// TIA Portal project "TaskCiclico" (V16)

(* hardware
DEVICE "S7-1200 station_1"  S7-1200 Station
   slot 0: "Telaio di montaggio_0"  S7-1200 Rack  Rack  V1.0
   slot 1: "PLC_1"  CPU 1214C DC/DC/DC  6ES7 214-1AG40-0XB0  V4.1
*)

// ===== PLC "PLC_1"  CPU 1214C DC/DC/DC =====

VAR_GLOBAL   // PLC tag table "Tabella delle variabili standard"
   "Reset" AT %I0.0 : Bool;
END_VAR

DATA_BLOCK "VariabiliGlobali"   // DB1
{ S7_Optimized_Access := 'TRUE' }
VERSION : 0.1
   VAR RETAIN
      Signal : Real;
      DelayedSignal : Real;
      N_SMP : Int := 5;
      SignalThreshold : Real := 40.0;
   END_VAR
BEGIN
END_DATA_BLOCK

DATA_BLOCK "FB_Shift_DB"   // DB2
{ S7_Optimized_Access := 'TRUE' }
VERSION : 0.1
// stored: InstanceOfName FB_Shift
"FB_Shift"
BEGIN
END_DATA_BLOCK

FUNCTION_BLOCK "FB_Shift"   // FB1, LAD
{ S7_Optimized_Access := 'TRUE' }
VERSION : 0.1
   VAR_INPUT
      Ingresso : Real;
      N_SMP : Int;
      Restart : Bool;
   END_VAR
   VAR_OUTPUT
      Uscita : Real;
   END_VAR
   VAR RETAIN
      STORE : Array[0..19] of Real;
      indice_1 : Int;
      indice_2 : Int;
      sup : Int;
   END_VAR
BEGIN

REGION Network 1
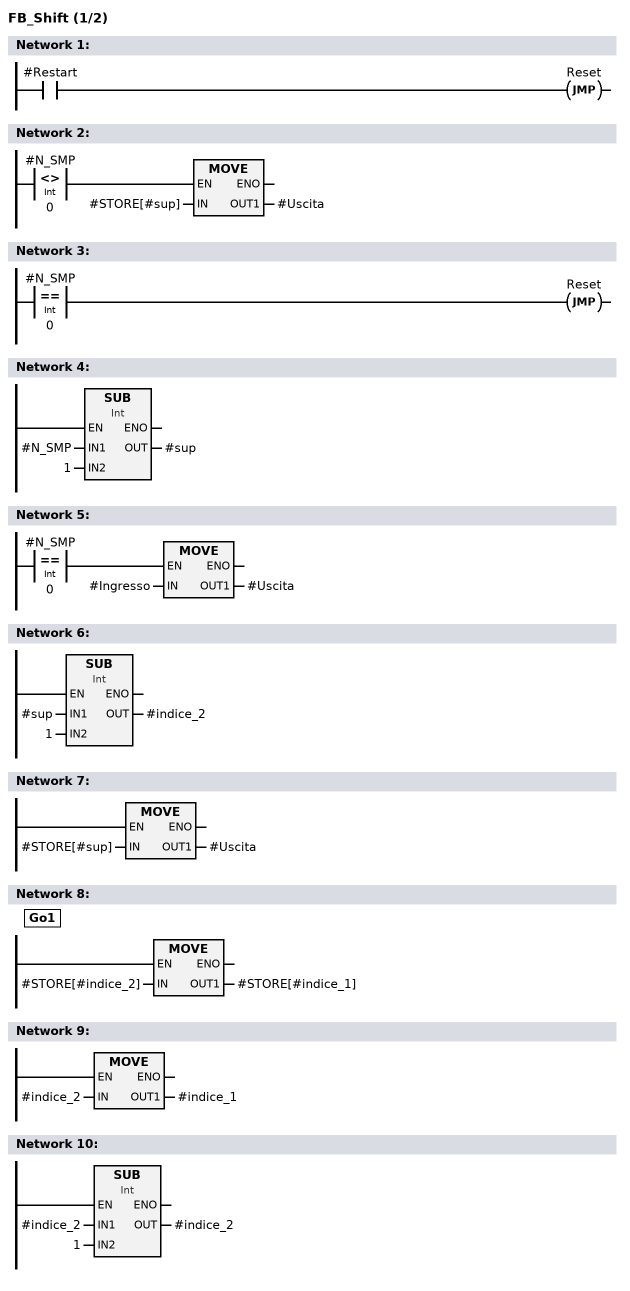
   RUNG wire#powerrail
      Contact( #Restart )
      JumpCoil( Reset )
   END_RUNG
   // the same network as SCL:
   IF #Restart THEN GOTO Reset; END_IF;
END_REGION

REGION Network 2
   RUNG wire#powerrail
      { S7_Templates := "SrcType := Int" } NE_Contact(in1 := #N_SMP, in2 := 0)
      Move(in := #STORE[#sup], out1 => #Uscita)
   END_RUNG
   // the same network as SCL:
   IF #N_SMP <> 0 THEN #Uscita := #STORE[#sup]; END_IF;
END_REGION

REGION Network 3
   RUNG wire#powerrail
      { S7_Templates := "SrcType := Int" } EQ_Contact(in1 := #N_SMP, in2 := 0)
      JumpCoil( Reset )
   END_RUNG
   // the same network as SCL:
   IF #N_SMP = 0 THEN GOTO Reset; END_IF;
END_REGION

REGION Network 4
   RUNG wire#powerrail
      { S7_Templates := "SrcType := Int" } Sub(in1 := #N_SMP, in2 := 1, out => #sup)
   END_RUNG
   // the same network as SCL:
   #sup := #N_SMP - 1;
END_REGION

REGION Network 5
   RUNG wire#powerrail
      { S7_Templates := "SrcType := Int" } EQ_Contact(in1 := #N_SMP, in2 := 0)
      Move(in := #Ingresso, out1 => #Uscita)
   END_RUNG
   // the same network as SCL:
   IF #N_SMP = 0 THEN #Uscita := #Ingresso; END_IF;
END_REGION

REGION Network 6
   RUNG wire#powerrail
      { S7_Templates := "SrcType := Int" } Sub(in1 := #sup, in2 := 1, out => #indice_2)
   END_RUNG
   // the same network as SCL:
   #indice_2 := #sup - 1;
END_REGION

REGION Network 7
   RUNG wire#powerrail
      { S7_GenerateENO := "TRUE" } Move(in := #STORE[#sup], out1 => #Uscita)
   END_RUNG
   // the same network as SCL:
   #Uscita := #STORE[#sup];
END_REGION

REGION Network 8
   Label( Go1 )
   RUNG wire#powerrail
      { S7_GenerateENO := "TRUE" } Move(in := #STORE[#indice_2], out1 => #STORE[#indice_1])
   END_RUNG
   // the same network as SCL:
   Go1:
   #STORE[#indice_1] := #STORE[#indice_2];
END_REGION

REGION Network 9
   RUNG wire#powerrail
      { S7_GenerateENO := "TRUE" } Move(in := #indice_2, out1 => #indice_1)
   END_RUNG
   // the same network as SCL:
   #indice_1 := #indice_2;
END_REGION

REGION Network 10
   RUNG wire#powerrail
      { S7_Templates := "SrcType := Int" } Sub(in1 := #indice_2, in2 := 1, out => #indice_2)
   END_RUNG
   // the same network as SCL:
   #indice_2 := #indice_2 - 1;
END_REGION

REGION Network 11
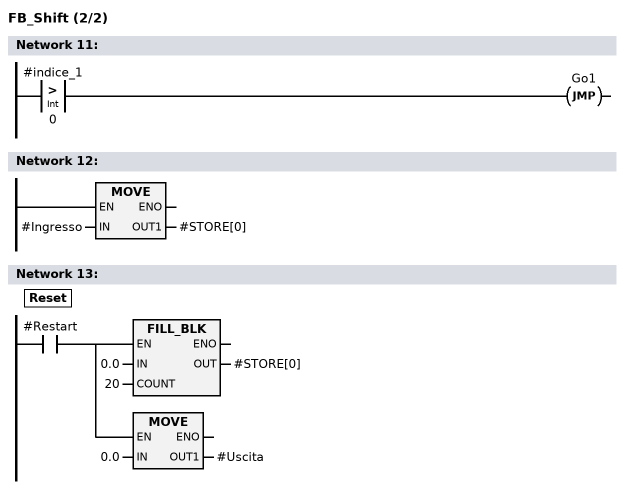
   RUNG wire#powerrail
      { S7_Templates := "SrcType := Int" } GT_Contact(in1 := #indice_1, in2 := 0)
      JumpCoil( Go1 )
   END_RUNG
   // the same network as SCL:
   IF #indice_1 > 0 THEN GOTO Go1; END_IF;
END_REGION

REGION Network 12
   RUNG wire#powerrail
      { S7_GenerateENO := "TRUE" } Move(in := #Ingresso, out1 => #STORE[0])
   END_RUNG
   // the same network as SCL:
   #STORE[0] := #Ingresso;
END_REGION

REGION Network 13
   Label( Reset )
   RUNG wire#powerrail
      Contact( #Restart )
      wire#w1
      FillBlockI(in := 0.0, count := 20, out => #STORE[0])
   END_RUNG
   RUNG wire#w1
      { S7_GenerateENO := "TRUE" } Move(in := 0.0, out1 => #Uscita)
   END_RUNG
   // the same network as SCL:
   Reset:
   IF #Restart THEN
       FILL_BLK(IN := 0.0, COUNT := 20, OUT => #STORE[0]);
       #Uscita := 0.0;
   END_IF;
END_REGION
END_FUNCTION_BLOCK

ORGANIZATION_BLOCK "Main"   // OB1, LAD, ProgramCycle
TITLE = "Main Program Sweep (Cycle)"
{ S7_Optimized_Access := 'TRUE' }
VERSION : 0.1
   VAR_INPUT
      Initial_Call : Bool;   // Initial call of this OB
      Remanence : Bool;   // =True, if remanent data are available
   END_VAR
BEGIN
END_ORGANIZATION_BLOCK

ORGANIZATION_BLOCK "Cyclic Task: Generatore Segnale"   // OB30, LAD, CyclicInterrupt
{ S7_Optimized_Access := 'TRUE' }
VERSION : 0.1
   VAR_INPUT
      Initial_Call : Bool;   // Initial call of this OB
      Event_Count : Int;   // Events discarded
   END_VAR
BEGIN

REGION Network 1
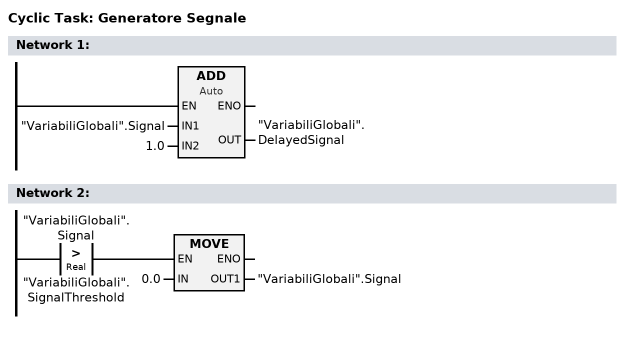
   RUNG wire#powerrail
      Add(in1 := "VariabiliGlobali".Signal, in2 := 1.0, out => "VariabiliGlobali".DelayedSignal)
   END_RUNG
   // the same network as SCL:
   "VariabiliGlobali".DelayedSignal := "VariabiliGlobali".Signal + 1.0;
END_REGION

REGION Network 2
   RUNG wire#powerrail
      { S7_Templates := "SrcType := Real" } GT_Contact(in1 := "VariabiliGlobali".Signal, in2 := "VariabiliGlobali".SignalThreshold)
      Move(in := 0.0, out1 => "VariabiliGlobali".Signal)
   END_RUNG
   // the same network as SCL:
   IF "VariabiliGlobali".Signal > "VariabiliGlobali".SignalThreshold THEN
       "VariabiliGlobali".Signal := 0.0;
   END_IF;
END_REGION
END_ORGANIZATION_BLOCK

ORGANIZATION_BLOCK "Cyclic Task: Richiamo FB Shift"   // OB31, LAD, CyclicInterrupt
{ S7_Optimized_Access := 'TRUE' }
VERSION : 0.1
   VAR_INPUT
      Initial_Call : Bool;   // Initial call of this OB
      Event_Count : Int;   // Events discarded
   END_VAR
BEGIN

REGION Network 1
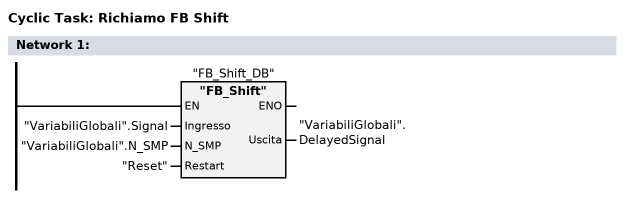
   RUNG wire#powerrail
      "FB_Shift_DB"(Ingresso := "VariabiliGlobali".Signal, N_SMP := "VariabiliGlobali".N_SMP, Restart := "Reset", Uscita => "VariabiliGlobali".DelayedSignal)
   END_RUNG
   // the same network as SCL:
   "FB_Shift_DB"(Ingresso := "VariabiliGlobali".Signal,   // "FB_Shift"
                 N_SMP := "VariabiliGlobali".N_SMP,
                 Restart := "Reset",
                 Uscita => "VariabiliGlobali".DelayedSignal);
END_REGION
END_ORGANIZATION_BLOCK